// TIA Portal V19 program export: 3 tag tables, 0 data types, 1 data blocks, 1 code blocks (in call order from the OBs), 0 instance data blocks

VAR_GLOBAL   // PLC tag table "Default tag table"
   System_Byte AT %MB101 : Byte;
   FirstScan AT %M101.0 : Bool;
   DiagStatusUpdate AT %M101.1 : Bool;
   AlwaysTRUE AT %M101.2 : Bool;
   AlwaysFALSE AT %M101.3 : Bool;
   Clock_Byte AT %MB100 : Byte;
   Clock_10Hz AT %M100.0 : Bool;
   Clock_5Hz AT %M100.1 : Bool;
   "Clock_2.5Hz" AT %M100.2 : Bool;
   Clock_2Hz AT %M100.3 : Bool;
   "Clock_1.25Hz" AT %M100.4 : Bool;
   Clock_1Hz AT %M100.5 : Bool;
   "Clock_0.625Hz" AT %M100.6 : Bool;
   "Clock_0.5Hz" AT %M100.7 : Bool;
   IW0For1500 AT %IW0 : Word;
   "InputData for 1500" AT %QW4 : Word;
   "1200POT_to_1500" AT %QW6 : Int;
END_VAR

VAR_GLOBAL   // PLC tag table "Comm with 1500"
   Green_from_1500 AT %M0.5 : Bool;
   Red_from_1500 AT %M0.6 : Bool;
   Blue_from_1500 AT %M0.7 : Bool;
   PB_Green_from_1500 AT %M0.0 : Bool;
   PB_Blue_from_1500 AT %M0.1 : Bool;
   OS1 AT %M2.0 : Bool;
   Error1 AT %M2.1 : Bool;
   status1 AT %MW4 : Word;
   history1 AT %MW6 : Word;
   Output_data_from_1500 AT %MB0 : Byte;
   OutputDataFrom1500 AT %MW0 : Word;
   Tag_6 AT %MW52 : Int;
   Input_buffer_to_1500 AT %MD50 : DWord;
END_VAR

VAR_GLOBAL   // PLC tag table "DemoCase"
   PB_Green_1200 AT %I0.0 : Bool;
   PB_Green_Lamp_1200 AT %Q0.0 : Bool;
   PB_Blue_1200 AT %I0.1 : Bool;
   PB_Blue_Lamp_1200 AT %Q0.1 : Bool;
   TopLights_Green_1200 AT %Q0.5 : Bool;
   TopLights_Red_1200 AT %Q0.6 : Bool;
   TopLights_Blue_1200 AT %Q0.7 : Bool;
   POT3_Upper_1200 AT %IW64 : Int;
   DataFrom1500 AT %IW4 : Word;
   IDevice AT %IB4 : Byte;
END_VAR

DATA_BLOCK "Connect_DB"   // DB7
{ S7_Optimized_Access := 'TRUE' }
// stored: MemoryReserve 100
   VAR
      Send_C_connect { S7_SetPoint := 'True'} : TCON_Param;
      Rec_C_connect { S7_SetPoint := 'True'} : TCON_Param;
   END_VAR
BEGIN
   Send_C_connect.ID := 100;
   Send_C_connect.ACTIVE_EST := false;
   Send_C_connect.LOCAL_TSAP_ID_LEN := 2;
   Send_C_connect.REM_STADDR_LEN := 0;
   Send_C_connect.REM_TSAP_ID_LEN := 0;
   Send_C_connect.LOCAL_TSAP_ID[1] := 16#7;
   Send_C_connect.LOCAL_TSAP_ID[2] := 16#D1;
   Rec_C_connect.ID := 101;
   Rec_C_connect.ACTIVE_EST := false;
   Rec_C_connect.LOCAL_TSAP_ID_LEN := 2;
   Rec_C_connect.REM_SUBNET_ID_LEN := 0;
   Rec_C_connect.REM_STADDR_LEN := 0;
   Rec_C_connect.REM_TSAP_ID_LEN := 0;
   Rec_C_connect.LOCAL_TSAP_ID[1] := 16#7;
   Rec_C_connect.LOCAL_TSAP_ID[2] := 16#D0;
END_DATA_BLOCK

ORGANIZATION_BLOCK "Main"   // OB1, LAD, ProgramCycle
TITLE = "Main Program Sweep (Cycle)"
{ S7_Optimized_Access := 'TRUE' }
// stored: AutoNumber false, SetENOAutomatically false
BEGIN

REGION Network 1: Buffer inputs to send to 1500
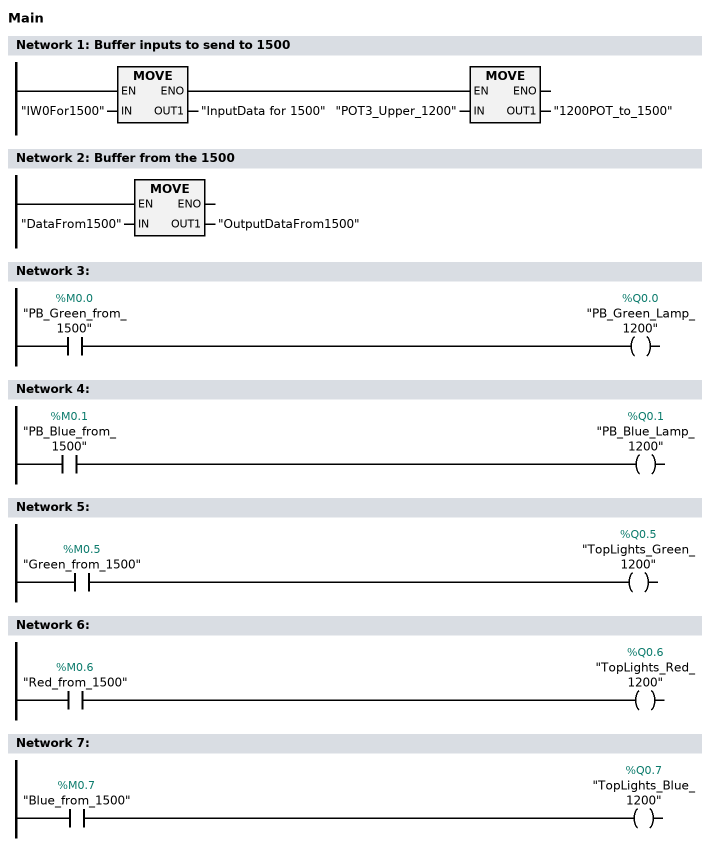
   RUNG wire#powerrail
      { S7_GenerateENO := "TRUE" } Move(in := "IW0For1500", out1 => "InputData for 1500")
      { S7_GenerateENO := "TRUE" } Move(in := "POT3_Upper_1200", out1 => "1200POT_to_1500")
   END_RUNG
   // the same network as SCL:
   // ENO of a box is taken as its EN; it also drops when the box reports an error
   "InputData for 1500" := "IW0For1500";
   "1200POT_to_1500" := "POT3_Upper_1200";
END_REGION

REGION Network 2: Buffer from the 1500
   RUNG wire#powerrail
      { S7_GenerateENO := "TRUE" } Move(in := "DataFrom1500", out1 => "OutputDataFrom1500")
   END_RUNG
   // the same network as SCL:
   "OutputDataFrom1500" := "DataFrom1500";
END_REGION

REGION Network 3
   RUNG wire#powerrail
      Contact( "PB_Green_from_1500" )
      Coil( "PB_Green_Lamp_1200" )
   END_RUNG
   // the same network as SCL:
   "PB_Green_Lamp_1200" := "PB_Green_from_1500";
END_REGION

REGION Network 4
   RUNG wire#powerrail
      Contact( "PB_Blue_from_1500" )
      Coil( "PB_Blue_Lamp_1200" )
   END_RUNG
   // the same network as SCL:
   "PB_Blue_Lamp_1200" := "PB_Blue_from_1500";
END_REGION

REGION Network 5
   RUNG wire#powerrail
      Contact( "Green_from_1500" )
      Coil( "TopLights_Green_1200" )
   END_RUNG
   // the same network as SCL:
   "TopLights_Green_1200" := "Green_from_1500";
END_REGION

REGION Network 6
   RUNG wire#powerrail
      Contact( "Red_from_1500" )
      Coil( "TopLights_Red_1200" )
   END_RUNG
   // the same network as SCL:
   "TopLights_Red_1200" := "Red_from_1500";
END_REGION

REGION Network 7
   RUNG wire#powerrail
      Contact( "Blue_from_1500" )
      Coil( "TopLights_Blue_1200" )
   END_RUNG
   // the same network as SCL:
   "TopLights_Blue_1200" := "Blue_from_1500";
END_REGION
END_ORGANIZATION_BLOCK
